% RSLogix 500 project 04. Automatic Sensor Calibration.RSS, saved by version 8.30.00.16 %
PROJECT "UNTITLED"    % processor: Bul.1763 MicroLogix 1100 Series B %

PROGRAM FILES
  LAD 2 "MAIN"  7 rungs
  LAD 3 "DIGITALIO"  3 rungs
  LAD 4 "CALIBRACAO"  23 rungs
  LAD 5 "CONTROL"  6 rungs
  LAD 6 "SAMPLING"  2 rungs

DATA FILES
  O0 OUTPUT  4 elements
  I1 INPUT  6 elements
  S2 STATUS  66 elements
  B3 BINARY  2 elements
  T4 TIMER  18 elements
  C5 COUNTER  2 elements
  R6 CONTROL  1 elements
  N7 INTEGER  20 elements
  F8 FLOAT  10 elements

LADDER 2 "MAIN"
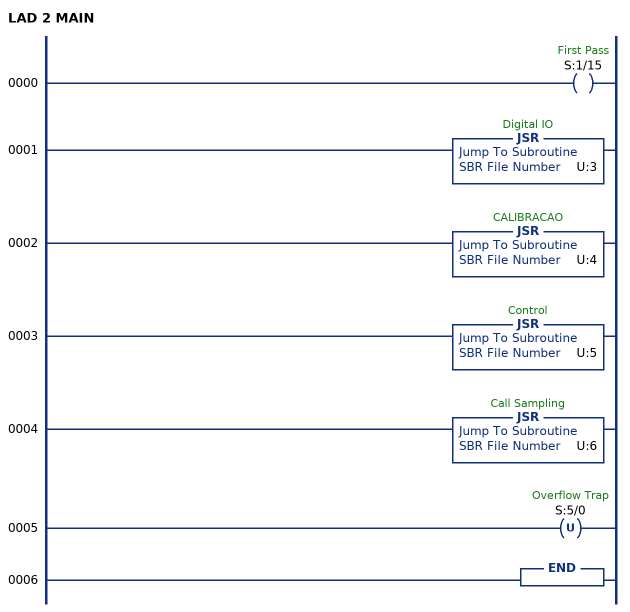
% Rung: 0 %
SOR OTE S:1/15 EOR
%   S:1/15  "First Pass" %
% Rung: 1 %
SOR JSR U:3 EOR
%   U:3  "Digital IO" %
% Rung: 2 %
SOR JSR U:4 EOR
%   U:4  "CALIBRACAO" %
% Rung: 3 %
SOR JSR U:5 EOR
%   U:5  "Control" %
% Rung: 4 %
SOR JSR U:6 EOR
%   U:6  "Call Sampling" %
% Rung: 5 %
SOR OTU S:5/0 EOR
%   S:5/0  "Overflow Trap" %
% Rung: 6 %
SOR END EOR

LADDER 3 "DIGITALIO"
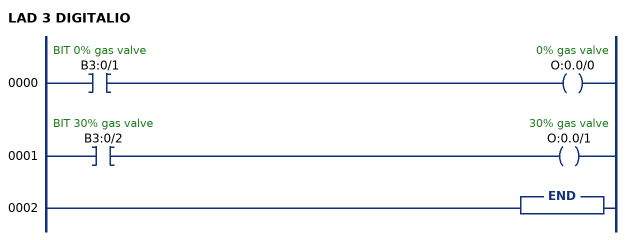
% Rung: 0 %
SOR XIC B3:0/1 OTE O:0.0/0 EOR
%   B3:0/1  "BIT 0% gas valve" %
%   O:0.0/0  "0% gas valve" %
% Rung: 1 %
SOR XIC B3:0/2 OTE O:0.0/1 EOR
%   B3:0/2  "BIT 30% gas valve" %
%   O:0.0/1  "30% gas valve" %
% Rung: 2 %
SOR END EOR

LADDER 4 "CALIBRACAO"
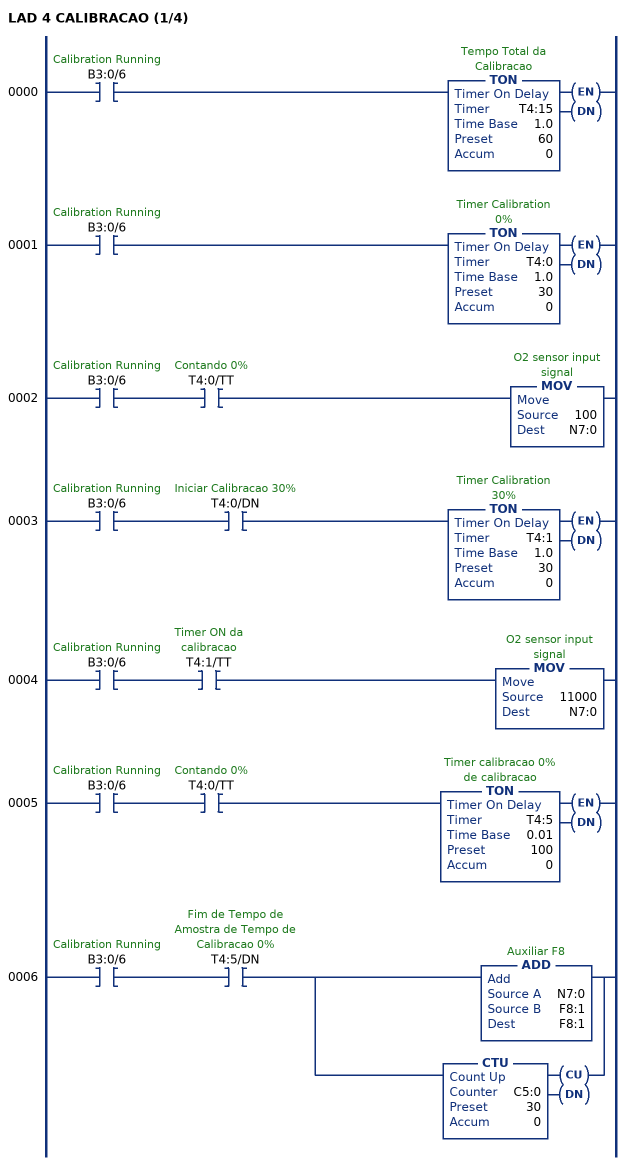
% Rung: 0 %
SOR XIC B3:0/6 TON T4:15 1.0 60 0 EOR
%   B3:0/6  "Calibration Running" %
%   T4:15  "Tempo Total da Calibracao" %
% Rung: 1 %
SOR XIC B3:0/6 TON T4:0 1.0 30 0 EOR
%   B3:0/6  "Calibration Running" %
%   T4:0  "Timer Calibration 0%" %
% Rung: 2 %
SOR XIC B3:0/6 XIC T4:0/TT MOV 100 N7:0 EOR
%   B3:0/6  "Calibration Running" %
%   T4:0/TT  "Contando 0%" %
%   N7:0  "O2 sensor input signal" %
% Rung: 3 %
SOR XIC B3:0/6 XIC T4:0/DN TON T4:1 1.0 30 0 EOR
%   B3:0/6  "Calibration Running" %
%   T4:0/DN  "Iniciar Calibracao 30%" %
%   T4:1  "Timer Calibration 30%" %
% Rung: 4 %
SOR XIC B3:0/6 XIC T4:1/TT MOV 11000 N7:0 EOR
%   B3:0/6  "Calibration Running" %
%   T4:1/TT  "Timer ON da calibracao" %
%   N7:0  "O2 sensor input signal" %
% Rung: 5 %
SOR XIC B3:0/6 XIC T4:0/TT TON T4:5 0.01 100 0 EOR
%   B3:0/6  "Calibration Running" %
%   T4:0/TT  "Contando 0%" %
%   T4:5  "Timer calibracao 0% de calibracao" %
% Rung: 6 %
SOR XIC B3:0/6 XIC T4:5/DN BST ADD N7:0 F8:1 F8:1 NXB CTU C5:0 30 0 BND EOR
%   B3:0/6  "Calibration Running" %
%   T4:5/DN  "Fim de Tempo de Amostra de Tempo de Calibracao 0%" %
%   N7:0  "O2 sensor input signal" %
%   F8:1  F8  "Auxiliar" %

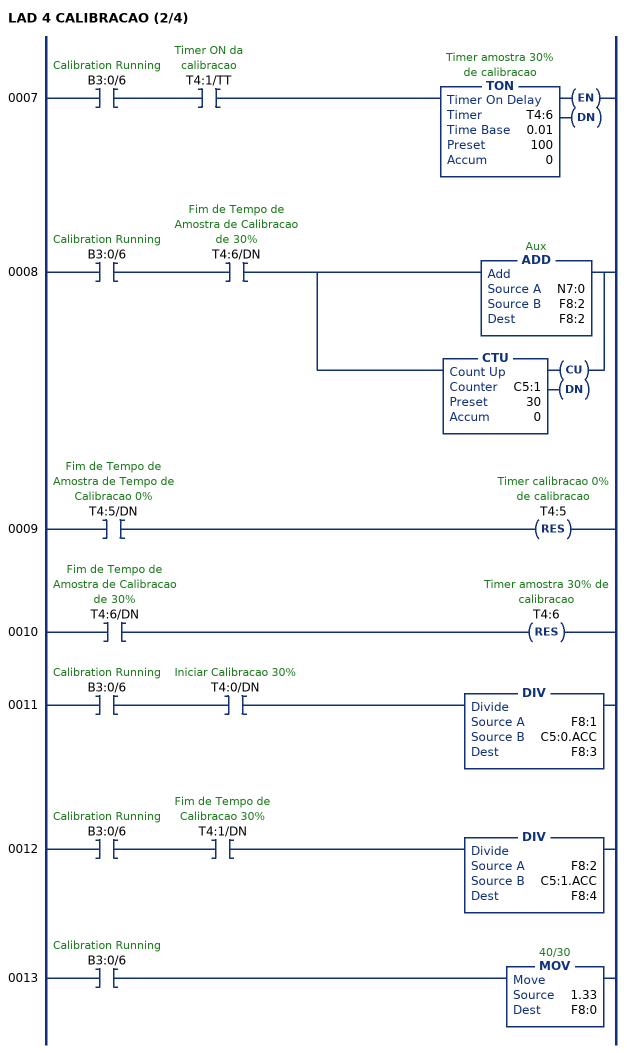
% Rung: 7 %
SOR XIC B3:0/6 XIC T4:1/TT TON T4:6 0.01 100 0 EOR
%   B3:0/6  "Calibration Running" %
%   T4:1/TT  "Timer ON da calibracao" %
%   T4:6  "Timer amostra 30% de calibracao" %
% Rung: 8 %
SOR XIC B3:0/6 XIC T4:6/DN BST ADD N7:0 F8:2 F8:2 NXB CTU C5:1 30 0 BND EOR
%   B3:0/6  "Calibration Running" %
%   T4:6/DN  "Fim de Tempo de Amostra de Calibracao de 30%" %
%   N7:0  "O2 sensor input signal" %
%   F8:2  "Aux" %
% Rung: 9 %
SOR XIC T4:5/DN RES T4:5 EOR
%   T4:5/DN  "Fim de Tempo de Amostra de Tempo de Calibracao 0%" %
%   T4:5  "Timer calibracao 0% de calibracao" %
% Rung: 10 %
SOR XIC T4:6/DN RES T4:6 EOR
%   T4:6/DN  "Fim de Tempo de Amostra de Calibracao de 30%" %
%   T4:6  "Timer amostra 30% de calibracao" %
% Rung: 11 %
SOR XIC B3:0/6 XIC T4:0/DN DIV F8:1 C5:0.ACC F8:3 EOR
%   B3:0/6  "Calibration Running" %
%   T4:0/DN  "Iniciar Calibracao 30%" %
%   F8:1  F8  "Auxiliar" %
% Rung: 12 %
SOR XIC B3:0/6 XIC T4:1/DN DIV F8:2 C5:1.ACC F8:4 EOR
%   B3:0/6  "Calibration Running" %
%   T4:1/DN  "Fim de Tempo de Calibracao 30%" %
%   F8:2  "Aux" %
% Rung: 13 %
SOR XIC B3:0/6 MOV 1.33 F8:0 EOR
%   B3:0/6  "Calibration Running" %
%   F8:0  "40/30" %

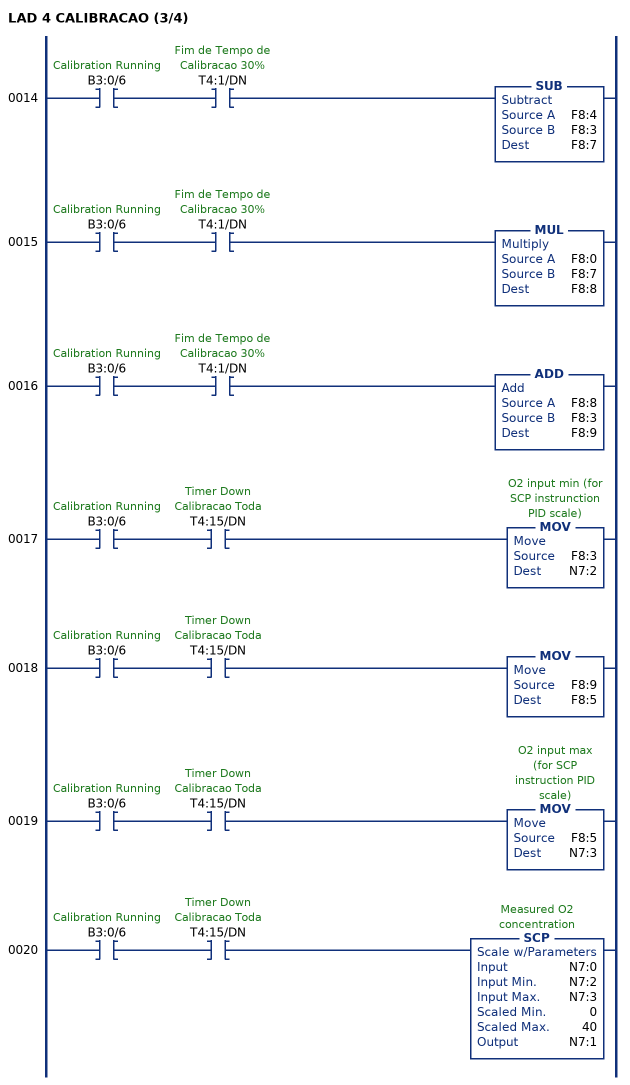
% Rung: 14 %
SOR XIC B3:0/6 XIC T4:1/DN SUB F8:4 F8:3 F8:7 EOR
%   B3:0/6  "Calibration Running" %
%   T4:1/DN  "Fim de Tempo de Calibracao 30%" %
% Rung: 15 %
SOR XIC B3:0/6 XIC T4:1/DN MUL F8:0 F8:7 F8:8 EOR
%   B3:0/6  "Calibration Running" %
%   T4:1/DN  "Fim de Tempo de Calibracao 30%" %
%   F8:0  "40/30" %
% Rung: 16 %
SOR XIC B3:0/6 XIC T4:1/DN ADD F8:8 F8:3 F8:9 EOR
%   B3:0/6  "Calibration Running" %
%   T4:1/DN  "Fim de Tempo de Calibracao 30%" %
% Rung: 17 %
SOR XIC B3:0/6 XIC T4:15/DN MOV F8:3 N7:2 EOR
%   B3:0/6  "Calibration Running" %
%   T4:15/DN  "Timer Down Calibracao Toda" %
%   N7:2  "O2 input min (for SCP instrunction PID scale)" %
% Rung: 18 %
SOR XIC B3:0/6 XIC T4:15/DN MOV F8:9 F8:5 EOR
%   B3:0/6  "Calibration Running" %
%   T4:15/DN  "Timer Down Calibracao Toda" %
% Rung: 19 %
SOR XIC B3:0/6 XIC T4:15/DN MOV F8:5 N7:3 EOR
%   B3:0/6  "Calibration Running" %
%   T4:15/DN  "Timer Down Calibracao Toda" %
%   N7:3  "O2 input max (for SCP instruction PID scale)" %
% Rung: 20 %
SOR XIC B3:0/6 XIC T4:15/DN SCP N7:0 N7:2 N7:3 0 40 N7:1 EOR
%   B3:0/6  "Calibration Running" %
%   T4:15/DN  "Timer Down Calibracao Toda" %
%   N7:0  "O2 sensor input signal" %
%   N7:2  "O2 input min (for SCP instrunction PID scale)" %
%   N7:3  "O2 input max (for SCP instruction PID scale)" %
%   N7:1  "Measured O2 concentration" %

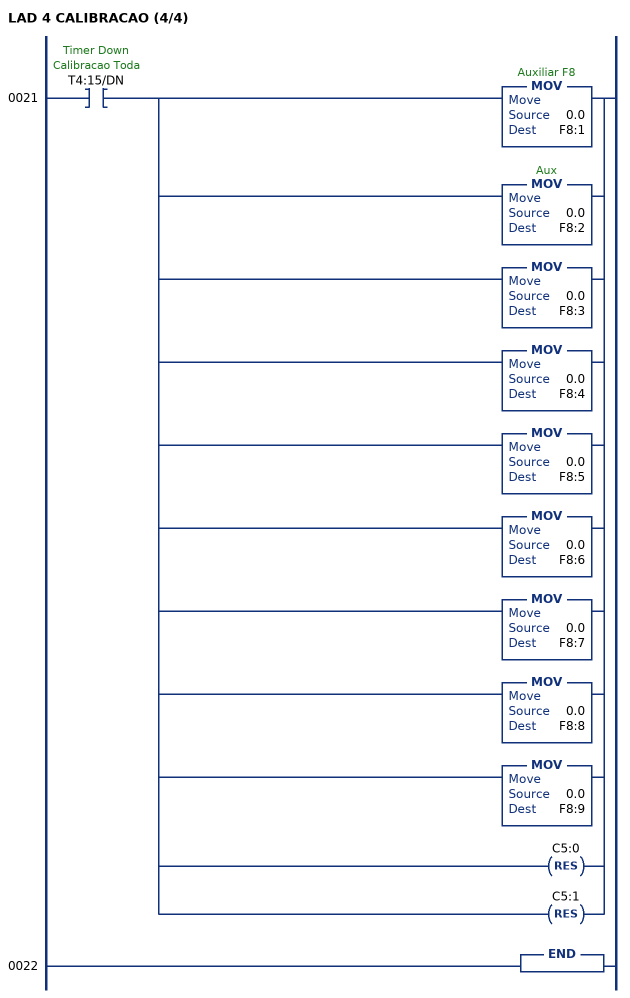
% Rung: 21 %
SOR XIC T4:15/DN BST MOV 0.0 F8:1 NXB MOV 0.0 F8:2 NXB MOV 0.0 F8:3 NXB MOV 0.0 F8:4 NXB MOV 0.0 F8:5 NXB MOV 0.0 F8:6 NXB MOV 0.0 F8:7 NXB MOV 0.0 F8:8 NXB MOV 0.0 F8:9 NXB RES C5:0 NXB RES C5:1 BND EOR
%   T4:15/DN  "Timer Down Calibracao Toda" %
%   F8:1  F8  "Auxiliar" %
%   F8:2  "Aux" %
% Rung: 22 %
SOR END EOR

LADDER 5 "CONTROL"
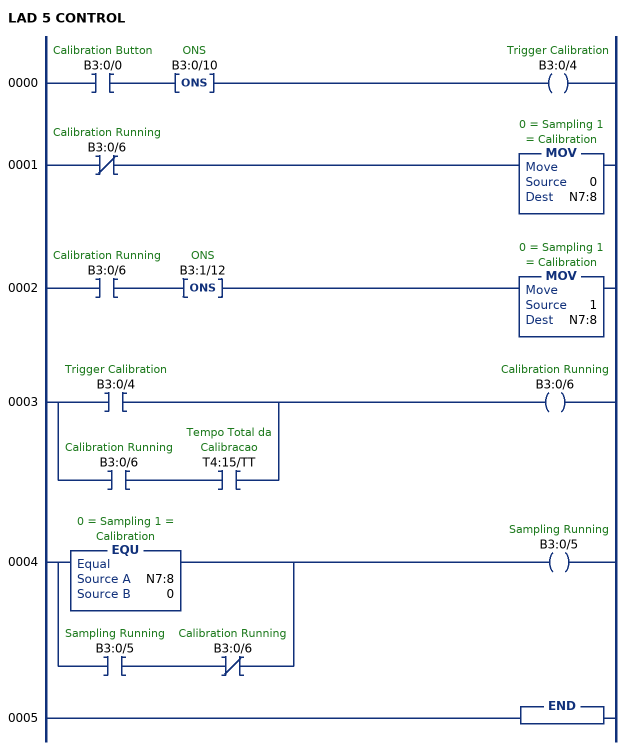
% Rung: 0 %
SOR XIC B3:0/0 ONS B3:0/10 OTE B3:0/4 EOR
%   B3:0/0  "Calibration Button" %
%   B3:0/10  "ONS" %
%   B3:0/4  "Trigger Calibration" %
% Rung: 1 %
SOR XIO B3:0/6 MOV 0 N7:8 EOR
%   B3:0/6  "Calibration Running" %
%   N7:8  "0 = Sampling 1 = Calibration" %
% Rung: 2 %
SOR XIC B3:0/6 ONS B3:1/12 MOV 1 N7:8 EOR
%   B3:0/6  "Calibration Running" %
%   B3:1/12  "ONS" %
%   N7:8  "0 = Sampling 1 = Calibration" %
% Rung: 3 %
SOR BST XIC B3:0/4 NXB XIC B3:0/6 XIC T4:15/TT BND OTE B3:0/6 EOR
%   B3:0/4  "Trigger Calibration" %
%   B3:0/6  "Calibration Running" %
%   T4:15/TT  "Tempo Total da Calibracao" %
% Rung: 4 %
SOR BST EQU N7:8 0 NXB XIC B3:0/5 XIO B3:0/6 BND OTE B3:0/5 EOR
%   N7:8  "0 = Sampling 1 = Calibration" %
%   B3:0/5  "Sampling Running" %
%   B3:0/6  "Calibration Running" %
% Rung: 5 %
SOR END EOR

LADDER 6 "SAMPLING"
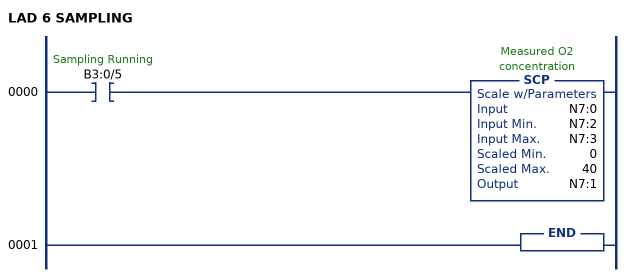
% Rung: 0 %
SOR XIC B3:0/5 SCP N7:0 N7:2 N7:3 0 40 N7:1 EOR
%   B3:0/5  "Sampling Running" %
%   N7:0  "O2 sensor input signal" %
%   N7:2  "O2 input min (for SCP instrunction PID scale)" %
%   N7:3  "O2 input max (for SCP instruction PID scale)" %
%   N7:1  "Measured O2 concentration" %
% Rung: 1 %
SOR END EOR

OTHER DOCUMENTED ADDRESSES
  B3:0/3  "Trigger Sampling"
  B3:0/7  "Sampling Button"
  B3:0/8  "Calibration Button"
  B3:0/9  "ONS"
  B3:1/0  "ONS"
  B3:1/1  "ONS"
  B3:1/2  "ONS"
  B3:1/3  "ONS"
  B3:1/4  "ONS"
  B3:1/5  "ONS"
  B3:1/6  "ONS"
  B3:1/7  "ONS"
  B3:1/10  "ONS"
  N7:0/0  "Abrindo valvula em 0%"
  N7:4  "Average 0% sampling"
  N7:5  "Average 30% sampling"
  N7:9  "Accumulado em Sampling Running"
  N7:10  "N7:10 = valor da media de amostra para Sampling Running"
  N7:11  "Acumulado Calibracao 0%"
  N7:12  "Acumulado calibracao 30%"
  N7:13  "Resultado da Calibracao 0%"
  N7:14  "Resultado Calibracao 30%"
  N7:15  "Input_Max"
  N7:16  "Auxiliar 01"
  N7:17  "Auxiliar 02"
  N7:18  "Auxiliar 03"
  N7:19  "Auxiliar 04"
  T4  "Reset Timer4"
  T4:3  "Sampling Time"
  T4:3/DN  "Acabou tempo de uma amostra"
  T4:4  "Tempo 30s de sampling"
  T4:4/TT  "Contando tempo de amostra"
  T4:16  "TimerAuxiliar"
  T4:16/TT  "Reset"
  T4:17  "TimerAuxiliar"
  T4:17/TT  "Reset"

DATA TABLE (non-zero values as saved)
DATA B3
% B3:0 % 0X0421 0X0008
DATA T4
% .PRE .ACC %
% T4:0 % 30 0
% T4:1 % 30 0
% T4:3 % 1 0
% T4:4 % 30 0
% T4:5 % 100 0
% T4:6 % 100 0
% T4:15 % 60 0
% T4:16 % 100 100
% T4:17 % 100 100
DATA C5
% .PRE .ACC %
% C5:0 % 30 0
% C5:1 % 30 0
DATA N7
% N7:0 % 14633 40 100 14597 0 0 0 0 0 0
DATA F8
% F8:0 % 1.33 0 0 0 0
